Staubli VAL3: Control_Timer.pgx

public program Control_Timer(string x_sMess, num x_nTime)
  local num l_nNow
begin
  //显示多长时间后消失
  call Control_PanelMd(x_sMess)
  l_nNow=clock()
  while clock()-l_nNow<=x_nTime
    delay(0)
  endWhile

end
